// TIA Portal V16 export
// export: Created 2024-09-05T17:39:13.3405005Z, ExportSetting WithDefaults, DisplayName Totally Integrated Automation Portal, DisplayVersion V16 Update 6, DisplayName TIA Portal Version Control Interface, DisplayVersion V16 Update 2, DisplayName TIA Portal Openness, DisplayVersion V16 Update 6, DisplayName STEP 7 Professional, DisplayVersion V16 Update 6, DisplayName STEP 7 Safety, DisplayVersion V16, DisplayName WinCC Advanced, DisplayVersion V16 Update 6
FUNCTION "READERS" : Void   // FC19, LAD
{ S7_Optimized_Access := 'TRUE' }
VERSION : 0.1
// stored: AutoNumber true, IsIECCheckEnabled false, SetENOAutomatically false, UDAEnableTagReadback false
   VAR_TEMP
      done1 : Bool;
      done2 : Bool;
      done3 : Bool;
      done4 : Bool;
      ERROR_RECIBIDO_ESCANER_REAR_TUBE : Int;
      ERROR_RECIBIDO_ESCANER_FRONT_TUBE : Int;
      ERROR_RECIBIDO_ESCANER_LH_MEMBER : Int;
      ERROR_RECIBIDO_ESCANER_RH_MEMBER : Int;
   END_VAR
   VAR_TEMP   // added for the SCL form of the ladder/FBD networks
      _w1 : Bool;
   END_VAR
BEGIN

REGION Network 1: INIT
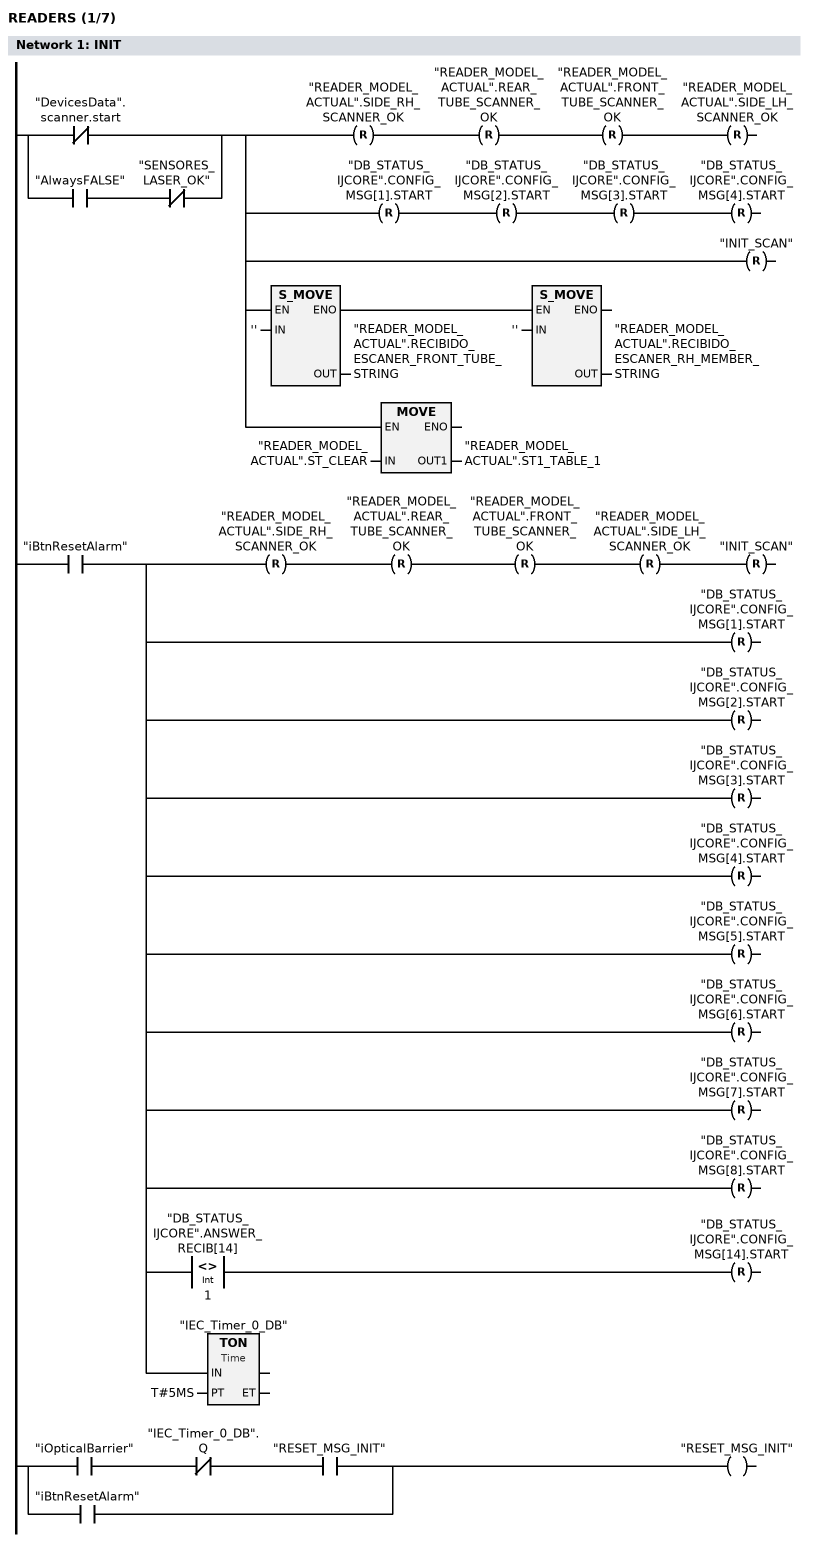
   RUNG wire#powerrail
      I_Contact( "DevicesData".scanner.start )
      wire#w1
      R_Coil( "READER_MODEL_ACTUAL".SIDE_RH_SCANNER_OK )
      R_Coil( "READER_MODEL_ACTUAL".REAR_TUBE_SCANNER_OK )
      R_Coil( "READER_MODEL_ACTUAL".FRONT_TUBE_SCANNER_OK )
      R_Coil( "READER_MODEL_ACTUAL".SIDE_LH_SCANNER_OK )
   END_RUNG
   RUNG wire#powerrail
      Contact( "AlwaysFALSE" )
      I_Contact( "SENSORES_LASER_OK" )
   END_RUNG wire#w1
   RUNG wire#w1
      R_Coil( "DB_STATUS_IJCORE".CONFIG_MSG[1].START )
      R_Coil( "DB_STATUS_IJCORE".CONFIG_MSG[2].START )
      R_Coil( "DB_STATUS_IJCORE".CONFIG_MSG[3].START )
      R_Coil( "DB_STATUS_IJCORE".CONFIG_MSG[4].START )
   END_RUNG
   RUNG wire#w1
      R_Coil( "INIT_SCAN" )
   END_RUNG
   RUNG wire#w1
      S_Move(in := '', out => "READER_MODEL_ACTUAL".RECIBIDO_ESCANER_FRONT_TUBE_STRING)
      S_Move(in := '', out => "READER_MODEL_ACTUAL".RECIBIDO_ESCANER_RH_MEMBER_STRING)
   END_RUNG
   RUNG wire#w1
      Move(in := "READER_MODEL_ACTUAL".ST_CLEAR, out1 => "READER_MODEL_ACTUAL".ST1_TABLE_1)
   END_RUNG
   RUNG wire#powerrail
      Contact( "iBtnResetAlarm" )
      wire#w2
      R_Coil( "READER_MODEL_ACTUAL".SIDE_RH_SCANNER_OK )
      R_Coil( "READER_MODEL_ACTUAL".REAR_TUBE_SCANNER_OK )
      R_Coil( "READER_MODEL_ACTUAL".FRONT_TUBE_SCANNER_OK )
      R_Coil( "READER_MODEL_ACTUAL".SIDE_LH_SCANNER_OK )
      R_Coil( "INIT_SCAN" )
   END_RUNG
   RUNG wire#w2
      R_Coil( "DB_STATUS_IJCORE".CONFIG_MSG[1].START )
   END_RUNG
   RUNG wire#w2
      R_Coil( "DB_STATUS_IJCORE".CONFIG_MSG[2].START )
   END_RUNG
   RUNG wire#w2
      R_Coil( "DB_STATUS_IJCORE".CONFIG_MSG[3].START )
   END_RUNG
   RUNG wire#w2
      R_Coil( "DB_STATUS_IJCORE".CONFIG_MSG[4].START )
   END_RUNG
   RUNG wire#w2
      R_Coil( "DB_STATUS_IJCORE".CONFIG_MSG[5].START )
   END_RUNG
   RUNG wire#w2
      R_Coil( "DB_STATUS_IJCORE".CONFIG_MSG[6].START )
   END_RUNG
   RUNG wire#w2
      R_Coil( "DB_STATUS_IJCORE".CONFIG_MSG[7].START )
   END_RUNG
   RUNG wire#w2
      R_Coil( "DB_STATUS_IJCORE".CONFIG_MSG[8].START )
   END_RUNG
   RUNG wire#w2
      { S7_Templates := "SrcType := Int" } NE_Contact(in1 := "DB_STATUS_IJCORE".ANSWER_RECIB[14], in2 := 1)
      R_Coil( "DB_STATUS_IJCORE".CONFIG_MSG[14].START )
   END_RUNG
   RUNG wire#w2
      { S7_Templates := "time_type := Time" } "IEC_Timer_0_DB".TON(pt := T#5MS, et =>)
   END_RUNG
   RUNG wire#powerrail
      Contact( "iOpticalBarrier" )
      I_Contact( "IEC_Timer_0_DB".Q )
      Contact( "RESET_MSG_INIT" )
      wire#w3
      Coil( "RESET_MSG_INIT" )
   END_RUNG
   RUNG wire#powerrail
      Contact( "iBtnResetAlarm" )
   END_RUNG wire#w3
   // the same network as SCL:
   IF NOT "DevicesData".scanner.start OR ("AlwaysFALSE" AND NOT "SENSORES_LASER_OK") THEN
       "READER_MODEL_ACTUAL".SIDE_RH_SCANNER_OK := FALSE;
       "READER_MODEL_ACTUAL".REAR_TUBE_SCANNER_OK := FALSE;
       "READER_MODEL_ACTUAL".FRONT_TUBE_SCANNER_OK := FALSE;
       "READER_MODEL_ACTUAL".SIDE_LH_SCANNER_OK := FALSE;
       "DB_STATUS_IJCORE".CONFIG_MSG[1].START := FALSE;
       "DB_STATUS_IJCORE".CONFIG_MSG[2].START := FALSE;
       "DB_STATUS_IJCORE".CONFIG_MSG[3].START := FALSE;
       "DB_STATUS_IJCORE".CONFIG_MSG[4].START := FALSE;
       "INIT_SCAN" := FALSE;
       "READER_MODEL_ACTUAL".RECIBIDO_ESCANER_FRONT_TUBE_STRING := '';
       "READER_MODEL_ACTUAL".RECIBIDO_ESCANER_RH_MEMBER_STRING := '';
       "READER_MODEL_ACTUAL".ST1_TABLE_1 := "READER_MODEL_ACTUAL".ST_CLEAR;
   END_IF;
   IF "iBtnResetAlarm" THEN
       "READER_MODEL_ACTUAL".SIDE_RH_SCANNER_OK := FALSE;
       "READER_MODEL_ACTUAL".REAR_TUBE_SCANNER_OK := FALSE;
       "READER_MODEL_ACTUAL".FRONT_TUBE_SCANNER_OK := FALSE;
       "READER_MODEL_ACTUAL".SIDE_LH_SCANNER_OK := FALSE;
       "INIT_SCAN" := FALSE;
       "DB_STATUS_IJCORE".CONFIG_MSG[1].START := FALSE;
       "DB_STATUS_IJCORE".CONFIG_MSG[2].START := FALSE;
       "DB_STATUS_IJCORE".CONFIG_MSG[3].START := FALSE;
       "DB_STATUS_IJCORE".CONFIG_MSG[4].START := FALSE;
       "DB_STATUS_IJCORE".CONFIG_MSG[5].START := FALSE;
       "DB_STATUS_IJCORE".CONFIG_MSG[6].START := FALSE;
       "DB_STATUS_IJCORE".CONFIG_MSG[7].START := FALSE;
       "DB_STATUS_IJCORE".CONFIG_MSG[8].START := FALSE;
   END_IF;
   IF "iBtnResetAlarm" AND ("DB_STATUS_IJCORE".ANSWER_RECIB[14] <> 1) THEN
       "DB_STATUS_IJCORE".CONFIG_MSG[14].START := FALSE;
   END_IF;
   "IEC_Timer_0_DB".TON(IN := "iBtnResetAlarm", PT := T#5MS);
   "RESET_MSG_INIT" := ("iOpticalBarrier" AND NOT "IEC_Timer_0_DB".Q AND "RESET_MSG_INIT") OR "iBtnResetAlarm";
END_REGION

REGION Network 2: CHARGE DATA FOR MODEL
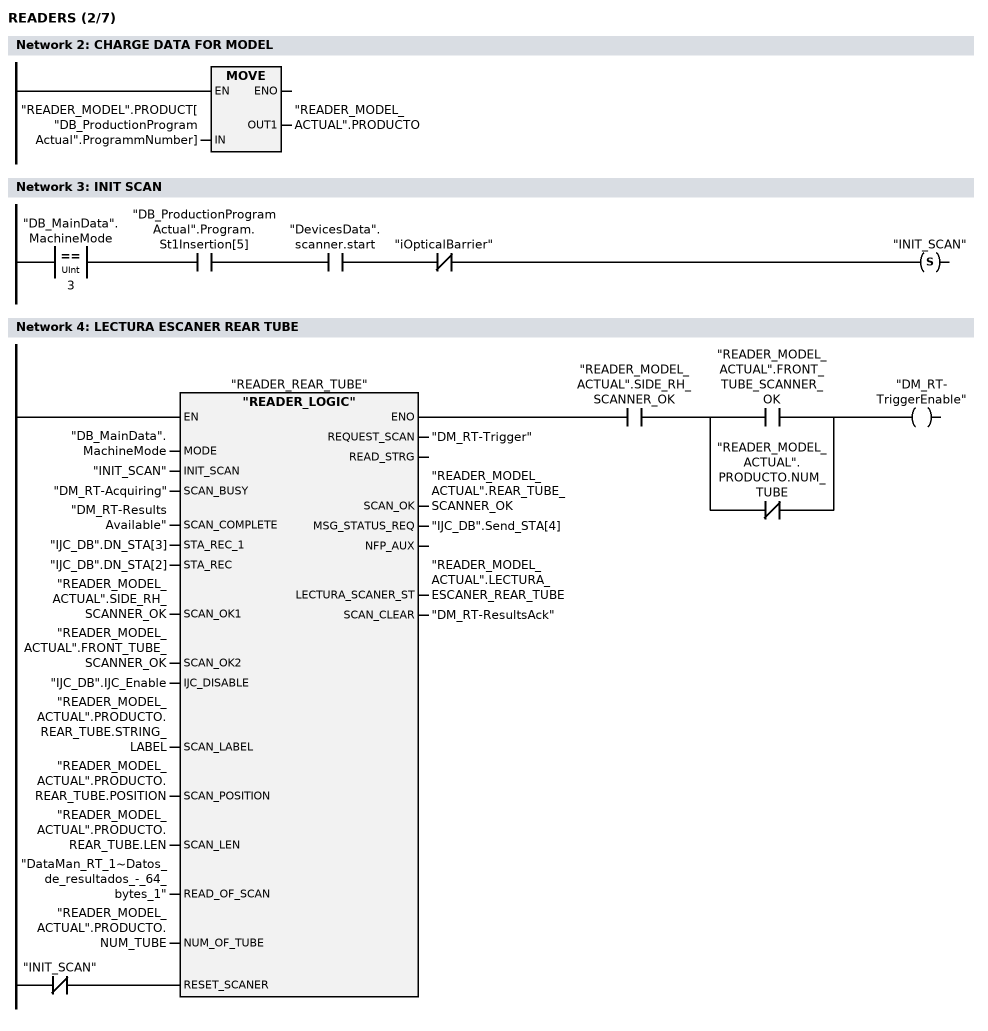
   RUNG wire#powerrail
      Move(in := "READER_MODEL".PRODUCT["DB_ProductionProgramActual".ProgrammNumber], out1 => "READER_MODEL_ACTUAL".PRODUCTO)
   END_RUNG
   // the same network as SCL:
   "READER_MODEL_ACTUAL".PRODUCTO := "READER_MODEL".PRODUCT["DB_ProductionProgramActual".ProgrammNumber];
END_REGION

REGION Network 3: INIT SCAN
   RUNG wire#powerrail
      { S7_Templates := "SrcType := UInt" } EQ_Contact(in1 := "DB_MainData".MachineMode, in2 := 3)
      Contact( "DB_ProductionProgramActual".Program.St1Insertion[5] )
      Contact( "DevicesData".scanner.start )
      I_Contact( "iOpticalBarrier" )
      S_Coil( "INIT_SCAN" )
   END_RUNG
   // the same network as SCL:
   IF ("DB_MainData".MachineMode = 3) AND "DB_ProductionProgramActual".Program.St1Insertion[5] AND "DevicesData".scanner.start AND NOT "iOpticalBarrier" THEN
       "INIT_SCAN" := TRUE;
   END_IF;
END_REGION

REGION Network 4: LECTURA ESCANER REAR TUBE
   RUNG wire#powerrail
      "READER_REAR_TUBE"(RESET_SCANER := wire#w1, MODE := "DB_MainData".MachineMode, INIT_SCAN := "INIT_SCAN", SCAN_BUSY := "DM_RT-Acquiring", SCAN_COMPLETE := "DM_RT-Results Available", STA_REC_1 := "IJC_DB".DN_STA[3], STA_REC := "IJC_DB".DN_STA[2], SCAN_OK1 := "READER_MODEL_ACTUAL".SIDE_RH_SCANNER_OK, SCAN_OK2 := "READER_MODEL_ACTUAL".FRONT_TUBE_SCANNER_OK, IJC_DISABLE := "IJC_DB".IJC_Enable, SCAN_LABEL := "READER_MODEL_ACTUAL".PRODUCTO.REAR_TUBE.STRING_LABEL, SCAN_POSITION := "READER_MODEL_ACTUAL".PRODUCTO.REAR_TUBE.POSITION, SCAN_LEN := "READER_MODEL_ACTUAL".PRODUCTO.REAR_TUBE.LEN, READ_OF_SCAN := "DataMan_RT_1~Datos_de_resultados_-_64_bytes_1", NUM_OF_TUBE := "READER_MODEL_ACTUAL".PRODUCTO.NUM_TUBE, REQUEST_SCAN => "DM_RT-Trigger", READ_STRG =>, SCAN_OK => "READER_MODEL_ACTUAL".REAR_TUBE_SCANNER_OK, MSG_STATUS_REQ => "IJC_DB".Send_STA[4], NFP_AUX =>, LECTURA_SCANER_ST => "READER_MODEL_ACTUAL".LECTURA_ESCANER_REAR_TUBE, SCAN_CLEAR => "DM_RT-ResultsAck")
      Contact( "READER_MODEL_ACTUAL".SIDE_RH_SCANNER_OK )
      wire#w2
      Contact( "READER_MODEL_ACTUAL".FRONT_TUBE_SCANNER_OK )
      wire#w3
      Coil( "DM_RT-TriggerEnable" )
   END_RUNG
   RUNG wire#powerrail
      I_Contact( "INIT_SCAN" )
   END_RUNG wire#w1
   RUNG wire#w2
      I_Contact( "READER_MODEL_ACTUAL".PRODUCTO.NUM_TUBE )
   END_RUNG wire#w3
   // the same network as SCL:
   "READER_REAR_TUBE"(MODE := "DB_MainData".MachineMode,   // "READER_LOGIC"
                      INIT_SCAN := "INIT_SCAN",
                      SCAN_BUSY := "DM_RT-Acquiring",
                      SCAN_COMPLETE := "DM_RT-Results Available",
                      STA_REC_1 := "IJC_DB".DN_STA[3],
                      STA_REC := "IJC_DB".DN_STA[2],
                      SCAN_OK1 := "READER_MODEL_ACTUAL".SIDE_RH_SCANNER_OK,
                      SCAN_OK2 := "READER_MODEL_ACTUAL".FRONT_TUBE_SCANNER_OK,
                      IJC_DISABLE := "IJC_DB".IJC_Enable,
                      SCAN_LABEL := "READER_MODEL_ACTUAL".PRODUCTO.REAR_TUBE.STRING_LABEL,
                      SCAN_POSITION := "READER_MODEL_ACTUAL".PRODUCTO.REAR_TUBE.POSITION,
                      SCAN_LEN := "READER_MODEL_ACTUAL".PRODUCTO.REAR_TUBE.LEN,
                      READ_OF_SCAN := "DataMan_RT_1~Datos_de_resultados_-_64_bytes_1",
                      NUM_OF_TUBE := "READER_MODEL_ACTUAL".PRODUCTO.NUM_TUBE,
                      RESET_SCANER := NOT "INIT_SCAN",
                      REQUEST_SCAN => "DM_RT-Trigger",
                      SCAN_OK => "READER_MODEL_ACTUAL".REAR_TUBE_SCANNER_OK,
                      MSG_STATUS_REQ => "IJC_DB".Send_STA[4],
                      LECTURA_SCANER_ST => "READER_MODEL_ACTUAL".LECTURA_ESCANER_REAR_TUBE,
                      SCAN_CLEAR => "DM_RT-ResultsAck",
                      ENO => #_w1);
   "DM_RT-TriggerEnable" := #_w1 AND "READER_MODEL_ACTUAL".SIDE_RH_SCANNER_OK AND ("READER_MODEL_ACTUAL".FRONT_TUBE_SCANNER_OK OR NOT "READER_MODEL_ACTUAL".PRODUCTO.NUM_TUBE);
END_REGION

REGION Network 5: LECTURA ESCANER FRONT TUBE
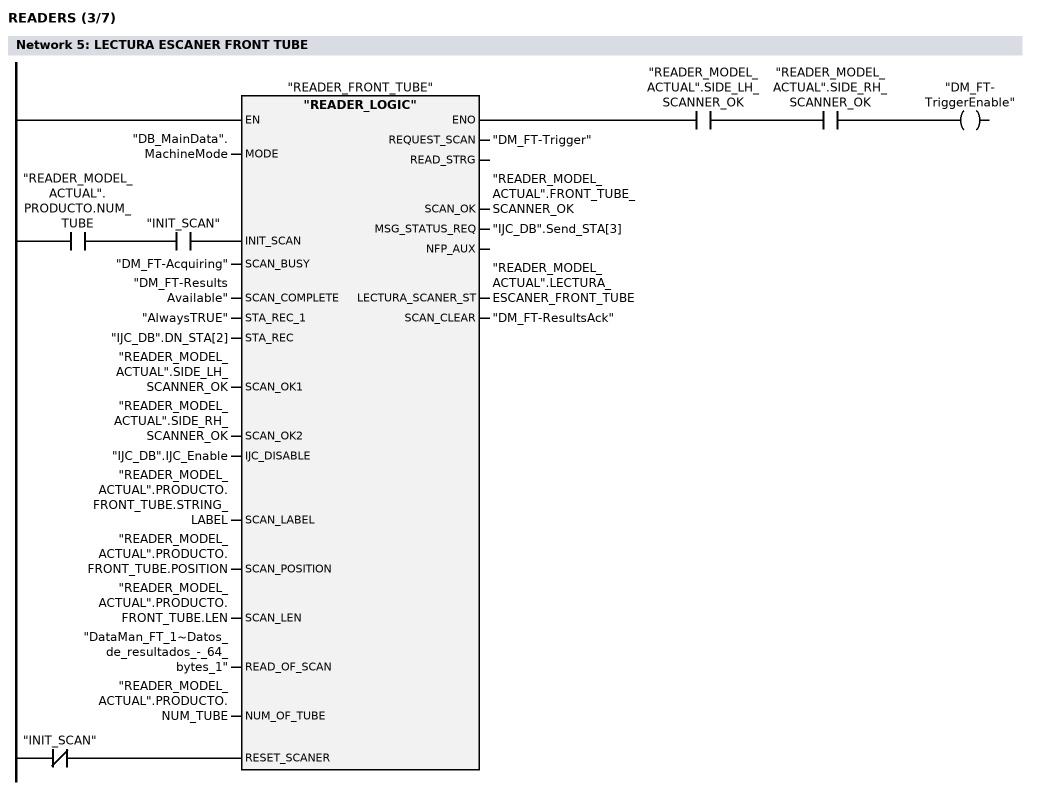
   RUNG wire#powerrail
      "READER_FRONT_TUBE"(INIT_SCAN := wire#w1, RESET_SCANER := wire#w2, MODE := "DB_MainData".MachineMode, SCAN_BUSY := "DM_FT-Acquiring", SCAN_COMPLETE := "DM_FT-Results Available", STA_REC_1 := "AlwaysTRUE", STA_REC := "IJC_DB".DN_STA[2], SCAN_OK1 := "READER_MODEL_ACTUAL".SIDE_LH_SCANNER_OK, SCAN_OK2 := "READER_MODEL_ACTUAL".SIDE_RH_SCANNER_OK, IJC_DISABLE := "IJC_DB".IJC_Enable, SCAN_LABEL := "READER_MODEL_ACTUAL".PRODUCTO.FRONT_TUBE.STRING_LABEL, SCAN_POSITION := "READER_MODEL_ACTUAL".PRODUCTO.FRONT_TUBE.POSITION, SCAN_LEN := "READER_MODEL_ACTUAL".PRODUCTO.FRONT_TUBE.LEN, READ_OF_SCAN := "DataMan_FT_1~Datos_de_resultados_-_64_bytes_1", NUM_OF_TUBE := "READER_MODEL_ACTUAL".PRODUCTO.NUM_TUBE, REQUEST_SCAN => "DM_FT-Trigger", READ_STRG =>, SCAN_OK => "READER_MODEL_ACTUAL".FRONT_TUBE_SCANNER_OK, MSG_STATUS_REQ => "IJC_DB".Send_STA[3], NFP_AUX =>, LECTURA_SCANER_ST => "READER_MODEL_ACTUAL".LECTURA_ESCANER_FRONT_TUBE, SCAN_CLEAR => "DM_FT-ResultsAck")
      Contact( "READER_MODEL_ACTUAL".SIDE_LH_SCANNER_OK )
      Contact( "READER_MODEL_ACTUAL".SIDE_RH_SCANNER_OK )
      Coil( "DM_FT-TriggerEnable" )
   END_RUNG
   RUNG wire#powerrail
      Contact( "READER_MODEL_ACTUAL".PRODUCTO.NUM_TUBE )
      Contact( "INIT_SCAN" )
   END_RUNG wire#w1
   RUNG wire#powerrail
      I_Contact( "INIT_SCAN" )
   END_RUNG wire#w2
   // the same network as SCL:
   "READER_FRONT_TUBE"(MODE := "DB_MainData".MachineMode,   // "READER_LOGIC"
                       INIT_SCAN := "READER_MODEL_ACTUAL".PRODUCTO.NUM_TUBE AND "INIT_SCAN",
                       SCAN_BUSY := "DM_FT-Acquiring",
                       SCAN_COMPLETE := "DM_FT-Results Available",
                       STA_REC_1 := "AlwaysTRUE",
                       STA_REC := "IJC_DB".DN_STA[2],
                       SCAN_OK1 := "READER_MODEL_ACTUAL".SIDE_LH_SCANNER_OK,
                       SCAN_OK2 := "READER_MODEL_ACTUAL".SIDE_RH_SCANNER_OK,
                       IJC_DISABLE := "IJC_DB".IJC_Enable,
                       SCAN_LABEL := "READER_MODEL_ACTUAL".PRODUCTO.FRONT_TUBE.STRING_LABEL,
                       SCAN_POSITION := "READER_MODEL_ACTUAL".PRODUCTO.FRONT_TUBE.POSITION,
                       SCAN_LEN := "READER_MODEL_ACTUAL".PRODUCTO.FRONT_TUBE.LEN,
                       READ_OF_SCAN := "DataMan_FT_1~Datos_de_resultados_-_64_bytes_1",
                       NUM_OF_TUBE := "READER_MODEL_ACTUAL".PRODUCTO.NUM_TUBE,
                       RESET_SCANER := NOT "INIT_SCAN",
                       REQUEST_SCAN => "DM_FT-Trigger",
                       SCAN_OK => "READER_MODEL_ACTUAL".FRONT_TUBE_SCANNER_OK,
                       MSG_STATUS_REQ => "IJC_DB".Send_STA[3],
                       LECTURA_SCANER_ST => "READER_MODEL_ACTUAL".LECTURA_ESCANER_FRONT_TUBE,
                       SCAN_CLEAR => "DM_FT-ResultsAck",
                       ENO => #_w1);
   "DM_FT-TriggerEnable" := #_w1 AND "READER_MODEL_ACTUAL".SIDE_LH_SCANNER_OK AND "READER_MODEL_ACTUAL".SIDE_RH_SCANNER_OK;
END_REGION

REGION Network 6: LECTURA ESCANER SIDE LH
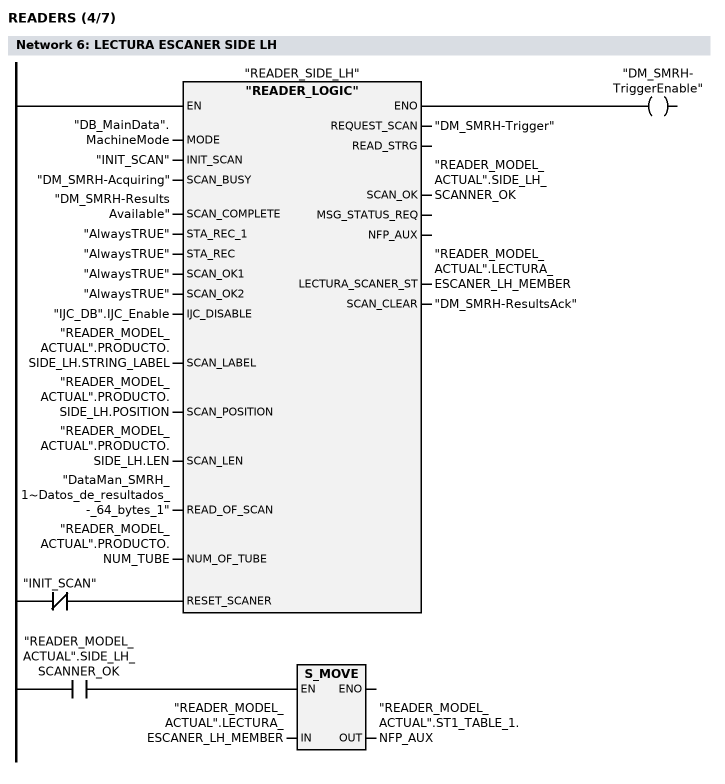
   RUNG wire#powerrail
      "READER_SIDE_LH"(RESET_SCANER := wire#w1, MODE := "DB_MainData".MachineMode, INIT_SCAN := "INIT_SCAN", SCAN_BUSY := "DM_SMRH-Acquiring", SCAN_COMPLETE := "DM_SMRH-Results Available", STA_REC_1 := "AlwaysTRUE", STA_REC := "AlwaysTRUE", SCAN_OK1 := "AlwaysTRUE", SCAN_OK2 := "AlwaysTRUE", IJC_DISABLE := "IJC_DB".IJC_Enable, SCAN_LABEL := "READER_MODEL_ACTUAL".PRODUCTO.SIDE_LH.STRING_LABEL, SCAN_POSITION := "READER_MODEL_ACTUAL".PRODUCTO.SIDE_LH.POSITION, SCAN_LEN := "READER_MODEL_ACTUAL".PRODUCTO.SIDE_LH.LEN, READ_OF_SCAN := "DataMan_SMRH_1~Datos_de_resultados_-_64_bytes_1", NUM_OF_TUBE := "READER_MODEL_ACTUAL".PRODUCTO.NUM_TUBE, REQUEST_SCAN => "DM_SMRH-Trigger", READ_STRG =>, SCAN_OK => "READER_MODEL_ACTUAL".SIDE_LH_SCANNER_OK, MSG_STATUS_REQ =>, NFP_AUX =>, LECTURA_SCANER_ST => "READER_MODEL_ACTUAL".LECTURA_ESCANER_LH_MEMBER, SCAN_CLEAR => "DM_SMRH-ResultsAck")
      Coil( "DM_SMRH-TriggerEnable" )
   END_RUNG
   RUNG wire#powerrail
      I_Contact( "INIT_SCAN" )
   END_RUNG wire#w1
   RUNG wire#powerrail
      Contact( "READER_MODEL_ACTUAL".SIDE_LH_SCANNER_OK )
      S_Move(in := "READER_MODEL_ACTUAL".LECTURA_ESCANER_LH_MEMBER, out => "READER_MODEL_ACTUAL".ST1_TABLE_1.NFP_AUX)
   END_RUNG
   // the same network as SCL:
   "READER_SIDE_LH"(MODE := "DB_MainData".MachineMode,   // "READER_LOGIC"
                    INIT_SCAN := "INIT_SCAN",
                    SCAN_BUSY := "DM_SMRH-Acquiring",
                    SCAN_COMPLETE := "DM_SMRH-Results Available",
                    STA_REC_1 := "AlwaysTRUE",
                    STA_REC := "AlwaysTRUE",
                    SCAN_OK1 := "AlwaysTRUE",
                    SCAN_OK2 := "AlwaysTRUE",
                    IJC_DISABLE := "IJC_DB".IJC_Enable,
                    SCAN_LABEL := "READER_MODEL_ACTUAL".PRODUCTO.SIDE_LH.STRING_LABEL,
                    SCAN_POSITION := "READER_MODEL_ACTUAL".PRODUCTO.SIDE_LH.POSITION,
                    SCAN_LEN := "READER_MODEL_ACTUAL".PRODUCTO.SIDE_LH.LEN,
                    READ_OF_SCAN := "DataMan_SMRH_1~Datos_de_resultados_-_64_bytes_1",
                    NUM_OF_TUBE := "READER_MODEL_ACTUAL".PRODUCTO.NUM_TUBE,
                    RESET_SCANER := NOT "INIT_SCAN",
                    REQUEST_SCAN => "DM_SMRH-Trigger",
                    SCAN_OK => "READER_MODEL_ACTUAL".SIDE_LH_SCANNER_OK,
                    LECTURA_SCANER_ST => "READER_MODEL_ACTUAL".LECTURA_ESCANER_LH_MEMBER,
                    SCAN_CLEAR => "DM_SMRH-ResultsAck",
                    ENO => #_w1);
   "DM_SMRH-TriggerEnable" := #_w1;
   IF "READER_MODEL_ACTUAL".SIDE_LH_SCANNER_OK THEN
       "READER_MODEL_ACTUAL".ST1_TABLE_1.NFP_AUX := "READER_MODEL_ACTUAL".LECTURA_ESCANER_LH_MEMBER;
   END_IF;
END_REGION

REGION Network 7: LECTURA ESCANER SIDE RH
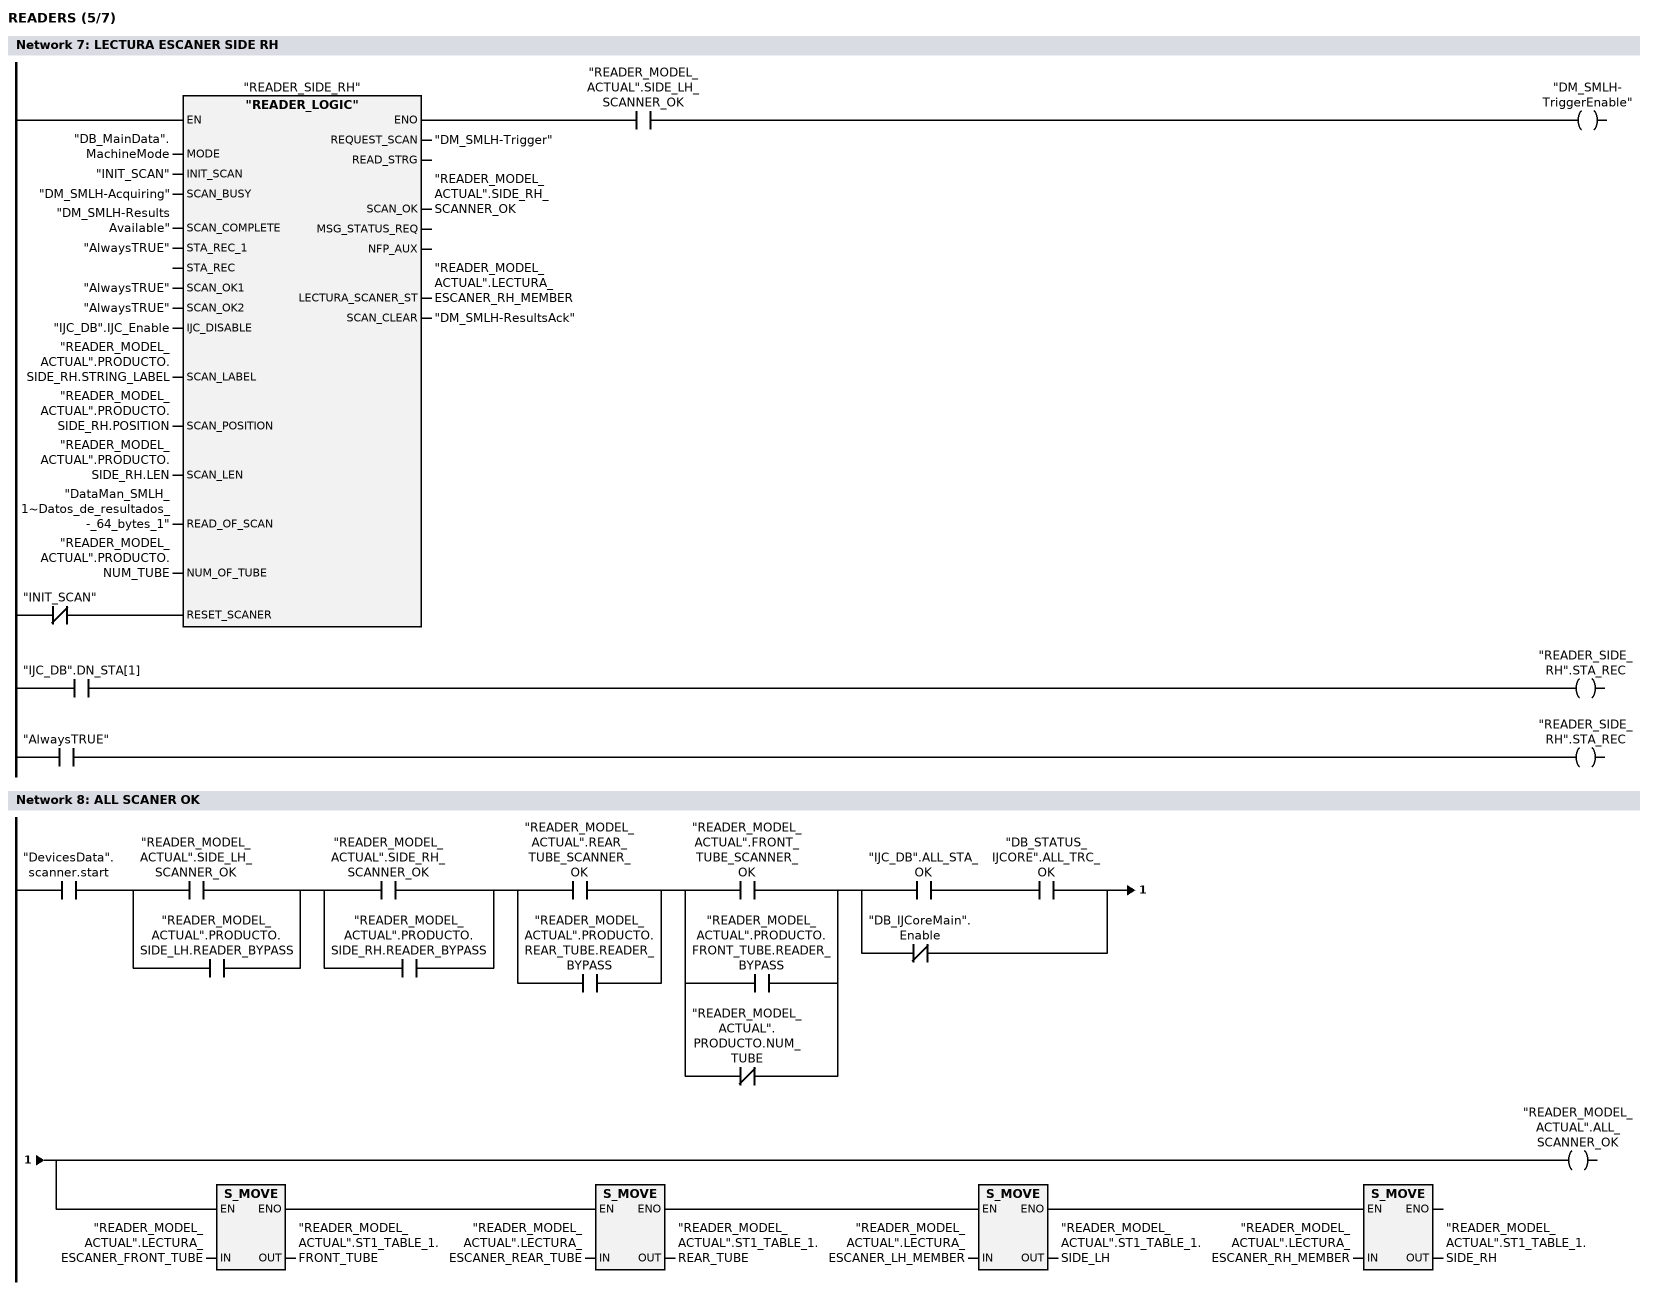
   RUNG wire#powerrail
      "READER_SIDE_RH"(RESET_SCANER := wire#w1, MODE := "DB_MainData".MachineMode, INIT_SCAN := "INIT_SCAN", SCAN_BUSY := "DM_SMLH-Acquiring", SCAN_COMPLETE := "DM_SMLH-Results Available", STA_REC_1 := "AlwaysTRUE", STA_REC :=, SCAN_OK1 := "AlwaysTRUE", SCAN_OK2 := "AlwaysTRUE", IJC_DISABLE := "IJC_DB".IJC_Enable, SCAN_LABEL := "READER_MODEL_ACTUAL".PRODUCTO.SIDE_RH.STRING_LABEL, SCAN_POSITION := "READER_MODEL_ACTUAL".PRODUCTO.SIDE_RH.POSITION, SCAN_LEN := "READER_MODEL_ACTUAL".PRODUCTO.SIDE_RH.LEN, READ_OF_SCAN := "DataMan_SMLH_1~Datos_de_resultados_-_64_bytes_1", NUM_OF_TUBE := "READER_MODEL_ACTUAL".PRODUCTO.NUM_TUBE, REQUEST_SCAN => "DM_SMLH-Trigger", READ_STRG =>, SCAN_OK => "READER_MODEL_ACTUAL".SIDE_RH_SCANNER_OK, MSG_STATUS_REQ =>, NFP_AUX =>, LECTURA_SCANER_ST => "READER_MODEL_ACTUAL".LECTURA_ESCANER_RH_MEMBER, SCAN_CLEAR => "DM_SMLH-ResultsAck")
      Contact( "READER_MODEL_ACTUAL".SIDE_LH_SCANNER_OK )
      Coil( "DM_SMLH-TriggerEnable" )
   END_RUNG
   RUNG wire#powerrail
      I_Contact( "INIT_SCAN" )
   END_RUNG wire#w1
   RUNG wire#powerrail
      Contact( "IJC_DB".DN_STA[1] )
      Coil( "READER_SIDE_RH".STA_REC )
   END_RUNG
   RUNG wire#powerrail
      Contact( "AlwaysTRUE" )
      Coil( "READER_SIDE_RH".STA_REC )
   END_RUNG
   // the same network as SCL:
   "READER_SIDE_RH"(MODE := "DB_MainData".MachineMode,   // "READER_LOGIC"
                    INIT_SCAN := "INIT_SCAN",
                    SCAN_BUSY := "DM_SMLH-Acquiring",
                    SCAN_COMPLETE := "DM_SMLH-Results Available",
                    STA_REC_1 := "AlwaysTRUE",
                    SCAN_OK1 := "AlwaysTRUE",
                    SCAN_OK2 := "AlwaysTRUE",
                    IJC_DISABLE := "IJC_DB".IJC_Enable,
                    SCAN_LABEL := "READER_MODEL_ACTUAL".PRODUCTO.SIDE_RH.STRING_LABEL,
                    SCAN_POSITION := "READER_MODEL_ACTUAL".PRODUCTO.SIDE_RH.POSITION,
                    SCAN_LEN := "READER_MODEL_ACTUAL".PRODUCTO.SIDE_RH.LEN,
                    READ_OF_SCAN := "DataMan_SMLH_1~Datos_de_resultados_-_64_bytes_1",
                    NUM_OF_TUBE := "READER_MODEL_ACTUAL".PRODUCTO.NUM_TUBE,
                    RESET_SCANER := NOT "INIT_SCAN",
                    REQUEST_SCAN => "DM_SMLH-Trigger",
                    SCAN_OK => "READER_MODEL_ACTUAL".SIDE_RH_SCANNER_OK,
                    LECTURA_SCANER_ST => "READER_MODEL_ACTUAL".LECTURA_ESCANER_RH_MEMBER,
                    SCAN_CLEAR => "DM_SMLH-ResultsAck",
                    ENO => #_w1);
   "DM_SMLH-TriggerEnable" := #_w1 AND "READER_MODEL_ACTUAL".SIDE_LH_SCANNER_OK;
   "READER_SIDE_RH".STA_REC := "IJC_DB".DN_STA[1];
   "READER_SIDE_RH".STA_REC := "AlwaysTRUE";
END_REGION

REGION Network 8: ALL SCANER OK
   RUNG wire#powerrail
      Contact( "DevicesData".scanner.start )
      wire#w1
      Contact( "READER_MODEL_ACTUAL".SIDE_LH_SCANNER_OK )
      wire#w2
      Contact( "READER_MODEL_ACTUAL".SIDE_RH_SCANNER_OK )
      wire#w3
      Contact( "READER_MODEL_ACTUAL".REAR_TUBE_SCANNER_OK )
      wire#w4
      Contact( "READER_MODEL_ACTUAL".FRONT_TUBE_SCANNER_OK )
      wire#w5
      Contact( "IJC_DB".ALL_STA_OK )
      Contact( "DB_STATUS_IJCORE".ALL_TRC_OK )
      wire#w6
      Coil( "READER_MODEL_ACTUAL".ALL_SCANNER_OK )
   END_RUNG
   RUNG wire#w1
      Contact( "READER_MODEL_ACTUAL".PRODUCTO.SIDE_LH.READER_BYPASS )
   END_RUNG wire#w2
   RUNG wire#w2
      Contact( "READER_MODEL_ACTUAL".PRODUCTO.SIDE_RH.READER_BYPASS )
   END_RUNG wire#w3
   RUNG wire#w3
      Contact( "READER_MODEL_ACTUAL".PRODUCTO.REAR_TUBE.READER_BYPASS )
   END_RUNG wire#w4
   RUNG wire#w4
      Contact( "READER_MODEL_ACTUAL".PRODUCTO.FRONT_TUBE.READER_BYPASS )
   END_RUNG wire#w5
   RUNG wire#w4
      I_Contact( "READER_MODEL_ACTUAL".PRODUCTO.NUM_TUBE )
   END_RUNG wire#w5
   RUNG wire#w5
      I_Contact( "DB_IJCoreMain".Enable )
   END_RUNG wire#w6
   RUNG wire#w6
      S_Move(in := "READER_MODEL_ACTUAL".LECTURA_ESCANER_FRONT_TUBE, out => "READER_MODEL_ACTUAL".ST1_TABLE_1.FRONT_TUBE)
      S_Move(in := "READER_MODEL_ACTUAL".LECTURA_ESCANER_REAR_TUBE, out => "READER_MODEL_ACTUAL".ST1_TABLE_1.REAR_TUBE)
      S_Move(in := "READER_MODEL_ACTUAL".LECTURA_ESCANER_LH_MEMBER, out => "READER_MODEL_ACTUAL".ST1_TABLE_1.SIDE_LH)
      S_Move(in := "READER_MODEL_ACTUAL".LECTURA_ESCANER_RH_MEMBER, out => "READER_MODEL_ACTUAL".ST1_TABLE_1.SIDE_RH)
   END_RUNG
   // the same network as SCL:
   "READER_MODEL_ACTUAL".ALL_SCANNER_OK := "DevicesData".scanner.start AND ("READER_MODEL_ACTUAL".SIDE_LH_SCANNER_OK OR "READER_MODEL_ACTUAL".PRODUCTO.SIDE_LH.READER_BYPASS) AND ("READER_MODEL_ACTUAL".SIDE_RH_SCANNER_OK OR "READER_MODEL_ACTUAL".PRODUCTO.SIDE_RH.READER_BYPASS) AND ("READER_MODEL_ACTUAL".REAR_TUBE_SCANNER_OK OR "READER_MODEL_ACTUAL".PRODUCTO.REAR_TUBE.READER_BYPASS) AND ("READER_MODEL_ACTUAL".FRONT_TUBE_SCANNER_OK OR "READER_MODEL_ACTUAL".PRODUCTO.FRONT_TUBE.READER_BYPASS OR NOT "READER_MODEL_ACTUAL".PRODUCTO.NUM_TUBE) AND (("IJC_DB".ALL_STA_OK AND "DB_STATUS_IJCORE".ALL_TRC_OK) OR NOT "DB_IJCoreMain".Enable);
   IF "READER_MODEL_ACTUAL".ALL_SCANNER_OK THEN
       "READER_MODEL_ACTUAL".ST1_TABLE_1.FRONT_TUBE := "READER_MODEL_ACTUAL".LECTURA_ESCANER_FRONT_TUBE;
       "READER_MODEL_ACTUAL".ST1_TABLE_1.REAR_TUBE := "READER_MODEL_ACTUAL".LECTURA_ESCANER_REAR_TUBE;
       "READER_MODEL_ACTUAL".ST1_TABLE_1.SIDE_LH := "READER_MODEL_ACTUAL".LECTURA_ESCANER_LH_MEMBER;
       "READER_MODEL_ACTUAL".ST1_TABLE_1.SIDE_RH := "READER_MODEL_ACTUAL".LECTURA_ESCANER_RH_MEMBER;
   END_IF;
END_REGION

REGION Network 9
   // "DB_ProductionProgramActual".Program.MechanicalType:
   // 0 - LH
   // 1 - RH
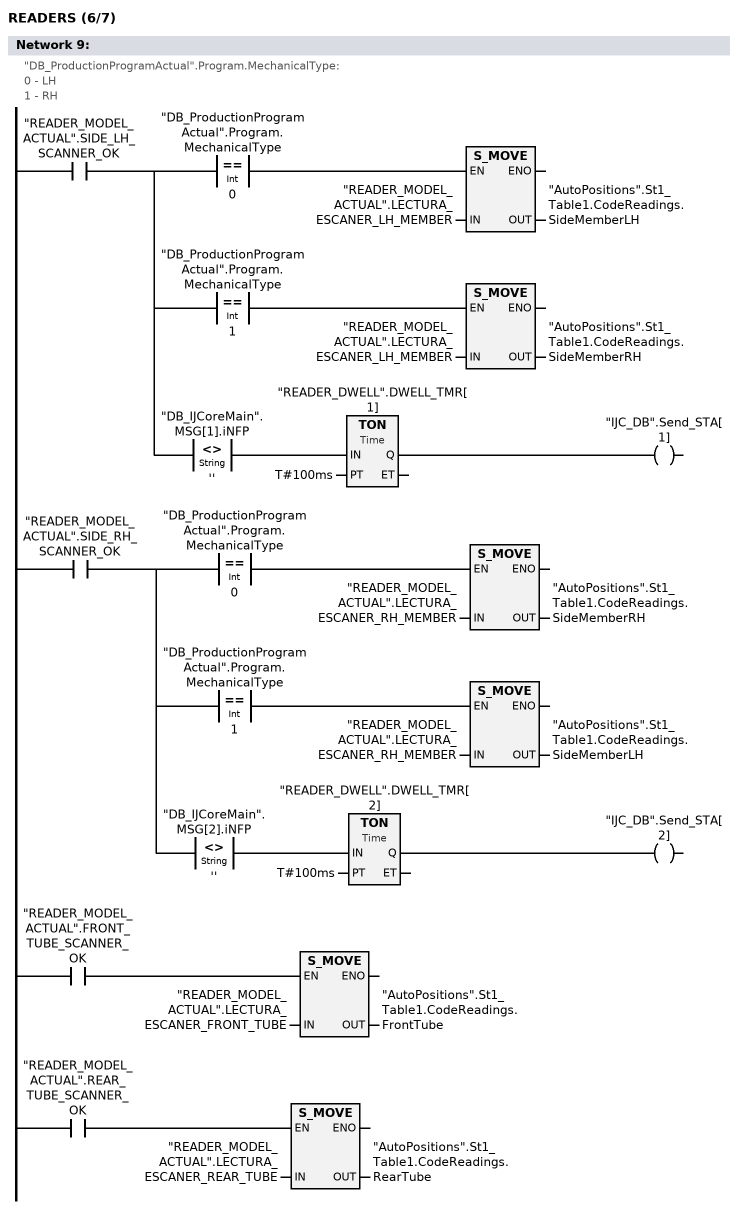
   RUNG wire#powerrail
      Contact( "READER_MODEL_ACTUAL".SIDE_LH_SCANNER_OK )
      wire#w1
      { S7_Templates := "SrcType := Int" } EQ_Contact(in1 := "DB_ProductionProgramActual".Program.MechanicalType, in2 := 0)
      S_Move(in := "READER_MODEL_ACTUAL".LECTURA_ESCANER_LH_MEMBER, out => "AutoPositions".St1_Table1.CodeReadings.SideMemberLH)
   END_RUNG
   RUNG wire#w1
      { S7_Templates := "SrcType := Int" } EQ_Contact(in1 := "DB_ProductionProgramActual".Program.MechanicalType, in2 := 1)
      S_Move(in := "READER_MODEL_ACTUAL".LECTURA_ESCANER_LH_MEMBER, out => "AutoPositions".St1_Table1.CodeReadings.SideMemberRH)
   END_RUNG
   RUNG wire#w1
      { S7_Templates := "SrcType := String" } NE_Contact(in1 := "DB_IJCoreMain".MSG[1].iNFP, in2 := '')
      { S7_Templates := "time_type := Time" } "READER_DWELL".DWELL_TMR[1].TON(pt := T#100ms, et =>)
      Coil( "IJC_DB".Send_STA[1] )
   END_RUNG
   RUNG wire#powerrail
      Contact( "READER_MODEL_ACTUAL".SIDE_RH_SCANNER_OK )
      wire#w2
      { S7_Templates := "SrcType := Int" } EQ_Contact(in1 := "DB_ProductionProgramActual".Program.MechanicalType, in2 := 0)
      S_Move(in := "READER_MODEL_ACTUAL".LECTURA_ESCANER_RH_MEMBER, out => "AutoPositions".St1_Table1.CodeReadings.SideMemberRH)
   END_RUNG
   RUNG wire#w2
      { S7_Templates := "SrcType := Int" } EQ_Contact(in1 := "DB_ProductionProgramActual".Program.MechanicalType, in2 := 1)
      S_Move(in := "READER_MODEL_ACTUAL".LECTURA_ESCANER_RH_MEMBER, out => "AutoPositions".St1_Table1.CodeReadings.SideMemberLH)
   END_RUNG
   RUNG wire#w2
      { S7_Templates := "SrcType := String" } NE_Contact(in1 := "DB_IJCoreMain".MSG[2].iNFP, in2 := '')
      { S7_Templates := "time_type := Time" } "READER_DWELL".DWELL_TMR[2].TON(pt := T#100ms, et =>)
      Coil( "IJC_DB".Send_STA[2] )
   END_RUNG
   RUNG wire#powerrail
      Contact( "READER_MODEL_ACTUAL".FRONT_TUBE_SCANNER_OK )
      S_Move(in := "READER_MODEL_ACTUAL".LECTURA_ESCANER_FRONT_TUBE, out => "AutoPositions".St1_Table1.CodeReadings.FrontTube)
   END_RUNG
   RUNG wire#powerrail
      Contact( "READER_MODEL_ACTUAL".REAR_TUBE_SCANNER_OK )
      S_Move(in := "READER_MODEL_ACTUAL".LECTURA_ESCANER_REAR_TUBE, out => "AutoPositions".St1_Table1.CodeReadings.RearTube)
   END_RUNG
   // the same network as SCL:
   IF "READER_MODEL_ACTUAL".SIDE_LH_SCANNER_OK AND ("DB_ProductionProgramActual".Program.MechanicalType = 0) THEN
       "AutoPositions".St1_Table1.CodeReadings.SideMemberLH := "READER_MODEL_ACTUAL".LECTURA_ESCANER_LH_MEMBER;
   END_IF;
   IF "READER_MODEL_ACTUAL".SIDE_LH_SCANNER_OK AND ("DB_ProductionProgramActual".Program.MechanicalType = 1) THEN
       "AutoPositions".St1_Table1.CodeReadings.SideMemberRH := "READER_MODEL_ACTUAL".LECTURA_ESCANER_LH_MEMBER;
   END_IF;
   "READER_DWELL".DWELL_TMR[1].TON(IN := "READER_MODEL_ACTUAL".SIDE_LH_SCANNER_OK AND ("DB_IJCoreMain".MSG[1].iNFP <> ''),
                           PT := T#100ms);
   "IJC_DB".Send_STA[1] := "READER_DWELL".DWELL_TMR[1].Q;
   IF "READER_MODEL_ACTUAL".SIDE_RH_SCANNER_OK AND ("DB_ProductionProgramActual".Program.MechanicalType = 0) THEN
       "AutoPositions".St1_Table1.CodeReadings.SideMemberRH := "READER_MODEL_ACTUAL".LECTURA_ESCANER_RH_MEMBER;
   END_IF;
   IF "READER_MODEL_ACTUAL".SIDE_RH_SCANNER_OK AND ("DB_ProductionProgramActual".Program.MechanicalType = 1) THEN
       "AutoPositions".St1_Table1.CodeReadings.SideMemberLH := "READER_MODEL_ACTUAL".LECTURA_ESCANER_RH_MEMBER;
   END_IF;
   "READER_DWELL".DWELL_TMR[2].TON(IN := "READER_MODEL_ACTUAL".SIDE_RH_SCANNER_OK AND ("DB_IJCoreMain".MSG[2].iNFP <> ''),
                           PT := T#100ms);
   "IJC_DB".Send_STA[2] := "READER_DWELL".DWELL_TMR[2].Q;
   IF "READER_MODEL_ACTUAL".FRONT_TUBE_SCANNER_OK THEN
       "AutoPositions".St1_Table1.CodeReadings.FrontTube := "READER_MODEL_ACTUAL".LECTURA_ESCANER_FRONT_TUBE;
   END_IF;
   IF "READER_MODEL_ACTUAL".REAR_TUBE_SCANNER_OK THEN
       "AutoPositions".St1_Table1.CodeReadings.RearTube := "READER_MODEL_ACTUAL".LECTURA_ESCANER_REAR_TUBE;
   END_IF;
END_REGION

REGION Network 10: SENSORES LASER
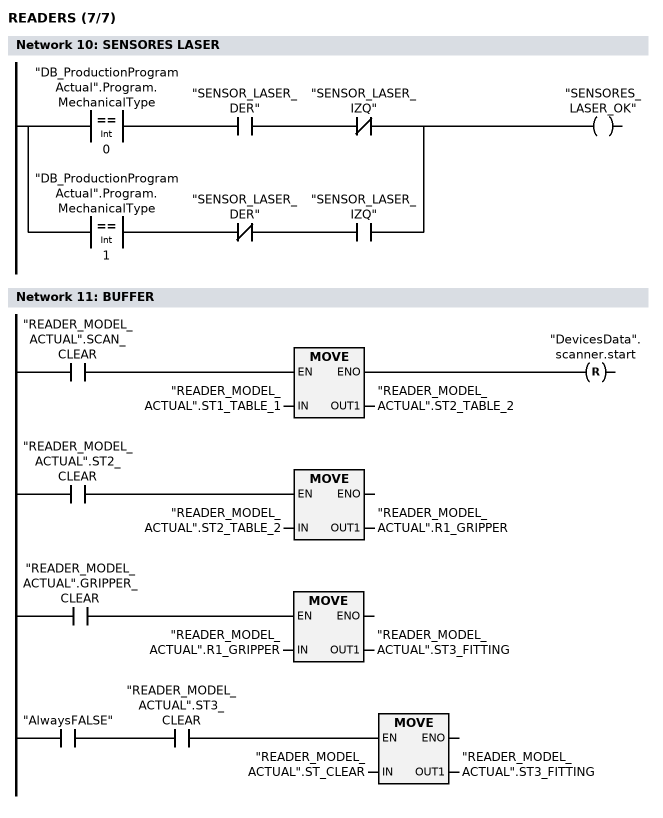
   RUNG wire#powerrail
      { S7_Templates := "SrcType := Int" } EQ_Contact(in1 := "DB_ProductionProgramActual".Program.MechanicalType, in2 := 0)
      Contact( "SENSOR_LASER_DER" )
      I_Contact( "SENSOR_LASER_IZQ" )
      wire#w1
      Coil( "SENSORES_LASER_OK" )
   END_RUNG
   RUNG wire#powerrail
      { S7_Templates := "SrcType := Int" } EQ_Contact(in1 := "DB_ProductionProgramActual".Program.MechanicalType, in2 := 1)
      I_Contact( "SENSOR_LASER_DER" )
      Contact( "SENSOR_LASER_IZQ" )
   END_RUNG wire#w1
   // the same network as SCL:
   "SENSORES_LASER_OK" := (("DB_ProductionProgramActual".Program.MechanicalType = 0) AND "SENSOR_LASER_DER" AND NOT "SENSOR_LASER_IZQ") OR (("DB_ProductionProgramActual".Program.MechanicalType = 1) AND NOT "SENSOR_LASER_DER" AND "SENSOR_LASER_IZQ");
END_REGION

REGION Network 11: BUFFER
   RUNG wire#powerrail
      Contact( "READER_MODEL_ACTUAL".SCAN_CLEAR )
      Move(in := "READER_MODEL_ACTUAL".ST1_TABLE_1, out1 => "READER_MODEL_ACTUAL".ST2_TABLE_2)
      R_Coil( "DevicesData".scanner.start )
   END_RUNG
   RUNG wire#powerrail
      Contact( "READER_MODEL_ACTUAL".ST2_CLEAR )
      Move(in := "READER_MODEL_ACTUAL".ST2_TABLE_2, out1 => "READER_MODEL_ACTUAL".R1_GRIPPER)
   END_RUNG
   RUNG wire#powerrail
      Contact( "READER_MODEL_ACTUAL".GRIPPER_CLEAR )
      Move(in := "READER_MODEL_ACTUAL".R1_GRIPPER, out1 => "READER_MODEL_ACTUAL".ST3_FITTING)
   END_RUNG
   RUNG wire#powerrail
      Contact( "AlwaysFALSE" )
      Contact( "READER_MODEL_ACTUAL".ST3_CLEAR )
      Move(in := "READER_MODEL_ACTUAL".ST_CLEAR, out1 => "READER_MODEL_ACTUAL".ST3_FITTING)
   END_RUNG
   // the same network as SCL:
   IF "READER_MODEL_ACTUAL".SCAN_CLEAR THEN
       "READER_MODEL_ACTUAL".ST2_TABLE_2 := "READER_MODEL_ACTUAL".ST1_TABLE_1;
       "DevicesData".scanner.start := FALSE;
   END_IF;
   IF "READER_MODEL_ACTUAL".ST2_CLEAR THEN
       "READER_MODEL_ACTUAL".R1_GRIPPER := "READER_MODEL_ACTUAL".ST2_TABLE_2;
   END_IF;
   IF "READER_MODEL_ACTUAL".GRIPPER_CLEAR THEN
       "READER_MODEL_ACTUAL".ST3_FITTING := "READER_MODEL_ACTUAL".R1_GRIPPER;
   END_IF;
   IF "AlwaysFALSE" AND "READER_MODEL_ACTUAL".ST3_CLEAR THEN
       "READER_MODEL_ACTUAL".ST3_FITTING := "READER_MODEL_ACTUAL".ST_CLEAR;
   END_IF;
END_REGION
END_FUNCTION
